FUNCTION TryConvert_DINT_TO_STRING : BOOL
VAR_INPUT
	in : DINT;
	out : REFERENCE TO STRING;
END_VAR

out := DINT_TO_STRING(in);
TryConvert_DINT_TO_STRING := TRUE;

END_FUNCTION

(* stored: Version 1.1.0.1, ProductVersion 3.1.4024.12
   POU TryConvert_DINT_TO_STRING: Id {0c4755b4-b919-4542-99f6-5e89fbe55a4b}, SpecialFunc None *)
